FUNCTION_BLOCK FB_RV
VAR_IN_OUT

END_VAR
VAR_INPUT
	Freigabe_auto			: BOOL;
	Freigabe_Deakt_auto		: BOOL;

	Betrieb_Anford_auto		: BOOL;

	Regelung_Modus_auto		: USINT;
	Regelung_Sollw_auto		: REAL;
	Regelung_Istw_auto		: REAL;

	Quittierung				: BOOL;
	Parameter_init			: ST_RV_Parameter;
END_VAR
VAR_OUTPUT
	{attribute 'OPC.UA.DA' := '1'}Parameter				: ST_RV_Parameter;	
	{attribute 'OPC.UA.DA' := '1'}Steuerung				: ST_RV_Steuerung;	
	{attribute 'OPC.UA.DA' := '1'}Stellwert				: ST_RV_Stellwert;	
	{attribute 'OPC.UA.DA' := '1'}Zustand					: ST_RV_Zustand;

END_VAR
VAR
	Zustandscheck			: FB_RV_Zustandscheck;
	Logik					: FB_RV_Logik;
	Ablaufsteuerung			: FB_RV_Ablaufsteuerung;
	Sollwertscheck			: FB_RV_Sollwertscheck;
	Regelung				: FB_RV_Regelung;
	Stellwertscheck			: FB_RV_Stellwertscheck;
	QuitTrig					: FB_SetResetFallTrigger;


	SchreibeDaten			: FB_RV_Output;
	OUT_Stellung			AT %Q* : INT;
	IN_Stellung				AT %I* : INT;
	Sollw_Test				: SINT;
END_VAR

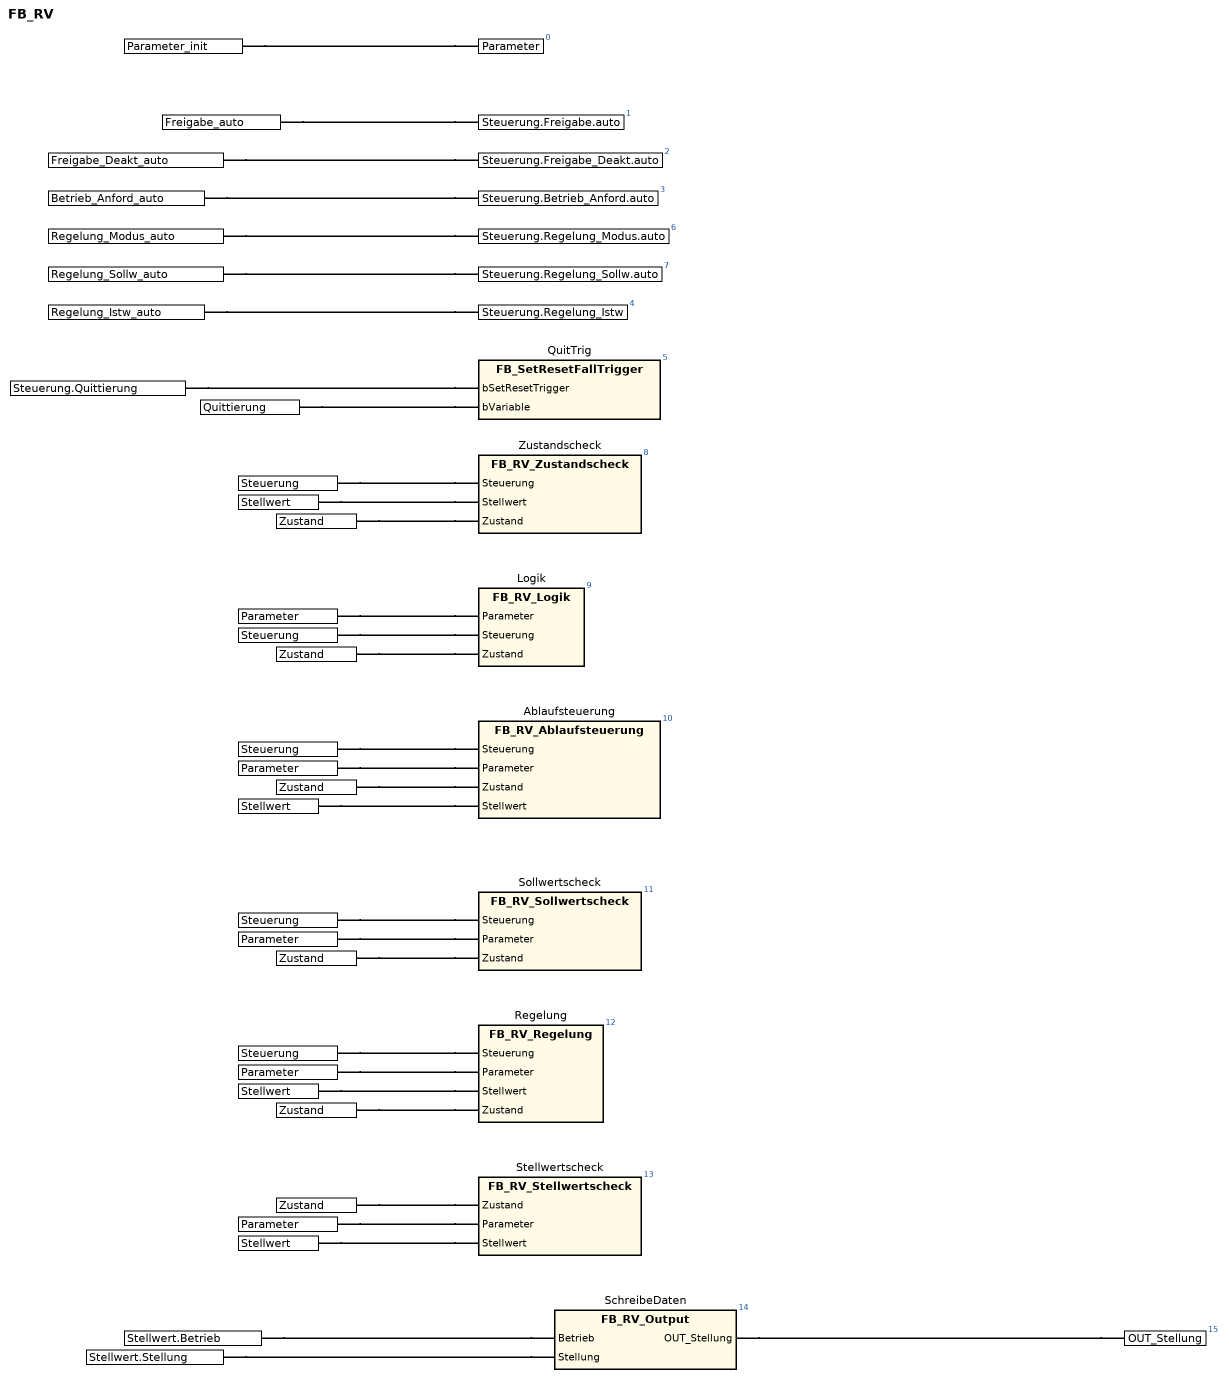
Parameter := Parameter_init;
Steuerung.Freigabe.auto := Freigabe_auto;
Steuerung.Freigabe_Deakt.auto := Freigabe_Deakt_auto;
Steuerung.Betrieb_Anford.auto := Betrieb_Anford_auto;
Steuerung.Regelung_Istw := Regelung_Istw_auto;
QuitTrig(bSetResetTrigger := Steuerung.Quittierung, bVariable := Quittierung); // FB_SetResetFallTrigger
Steuerung.Regelung_Modus.auto := Regelung_Modus_auto;
Steuerung.Regelung_Sollw.auto := Regelung_Sollw_auto;
Zustandscheck(Steuerung := Steuerung, Stellwert := Stellwert, Zustand := Zustand); // FB_RV_Zustandscheck
Logik(Parameter := Parameter, Steuerung := Steuerung, Zustand := Zustand); // FB_RV_Logik
Ablaufsteuerung(Steuerung := Steuerung, Parameter := Parameter, Zustand := Zustand, Stellwert := Stellwert); // FB_RV_Ablaufsteuerung
Sollwertscheck(Steuerung := Steuerung, Parameter := Parameter, Zustand := Zustand); // FB_RV_Sollwertscheck
Regelung(Steuerung := Steuerung, Parameter := Parameter, Stellwert := Stellwert, Zustand := Zustand); // FB_RV_Regelung
Stellwertscheck(Zustand := Zustand, Parameter := Parameter, Stellwert := Stellwert); // FB_RV_Stellwertscheck
SchreibeDaten(Betrieb := Stellwert.Betrieb, Stellung := Stellwert.Stellung); // FB_RV_Output
OUT_Stellung := SchreibeDaten.OUT_Stellung;

END_FUNCTION_BLOCK

(* stored: Version 1.1.0.1, ProductVersion 3.1.4024.9
   POU FB_RV: Id {9ee081b4-12af-4b2a-b1f2-e843636001ca}, SpecialFunc None *)
